FUNCTION_BLOCK FB_Blinker
VAR_INPUT
		bStart		:	BOOL;
	    tPeriode	:	TIME	:= T#1S;
END_VAR
VAR_OUTPUT
		bBlinker	: 	BOOL;
END_VAR
VAR
		fbTimer 	: 	TON;
END_VAR

fbTimer (IN:=bStart AND NOT fbTimer.Q, PT:= tPeriode,);

IF fbTimer.ET >= tPeriode/2
	THEN
	bBlinker:= TRUE;
	ELSE
	bBlinker:=FALSE;
	
END_IF

END_FUNCTION_BLOCK

(* stored: Version 1.1.0.1, ProductVersion 3.1.4024.3
   POU FB_Blinker: Id {bd16c604-cd72-4496-8744-1cb13084ac62}, SpecialFunc None *)
